Staubli VAL3: READTRAJ.pgx

public program ReadTraj()
  local bool l_bBool
begin
  TxtFile:bReadProduct=true
  if DataBase:nInterfaceType==5
    call TxtFile:ReadTraj("Disk://Txt/Recipe.txt",TxtFile:sProductName,nStartTraj,nEndTraj,l_bBool)
  else
    logMsg("读取"+"Disk://Txt/Product"+toString("",DataBase:nWorkPlaceIndex)+".txt")
    call TxtFile:ReadTraj("Disk://Txt/Product"+toString("",DataBase:nWorkPlaceIndex)+".txt",DataBase:sProductName[DataBase:nWorkPlaceIndex],1,TxtFile:nTotalTraj,l_bBool)
  endIf


  TxtFile:bReadProduct=false
  if !l_bBool
    disablePower()
    popUpMsg("读取路径信息出现异常")

    if DataBase:nInterfaceType==5
      logMsg(TxtFile:sProductName+"读取示教路径信息出现异常")
    else
      logMsg(DataBase:sProductName[DataBase:nWorkPlaceIndex]+"读取路径信息出现异常")
    endIf
  else
    //popUpMsg("读取路径OK")
  endIf



end
